Staubli VAL3: iPressureSensor.pgx

public program iPressureSensor(num& nNum[] (dimensions=1))
begin
  nNum=dioGet(iPressureSensor)
end
